FUNCTION_BLOCK "SEQUENCE"   // FB18, GRAPH_PLUS
{ S7_Optimized_Access := 'TRUE' }
VERSION : 0.1
   VAR_INPUT
      OFF_SQ : Bool := false;   // Turn sequence off
      INIT_SQ : Bool := false;   // Set sequence to initial state
      ACK_EF : Bool := false;   // Acknowledge all errors and faults
      S_PREV : Bool := false;   // Output previous step in parameter S_NO
      S_NEXT : Bool := false;   // Indicate next step in parameter S_NO
      SW_AUTO : Bool := false;   // Automatic mode
      SW_TAP : Bool := false;   // Semiautomatic/switch with transition
      SW_TOP : Bool := false;   // Semiautomatic/ignore transition
      SW_MAN : Bool := false;   // Manual mode
      S_SEL : Int := 0;   // Select step to be output to S_NO
      S_ON : Bool := false;   // Activate step indicated in S_NO
      S_OFF : Bool := false;   // Deactivate step indicated S_NO
      T_PUSH : Bool := false;   // Enable transition to switch in semi automatic mode
   END_VAR
   VAR_OUTPUT
      S_NO : Int := 0;   // Step number
      S_MORE : Bool := false;   // More steps are available and can be shown in S_NO
      S_ACTIVE : Bool := false;   // Step indicated in S_NO is active
      ERR_FLT : Bool := false;   // Interlock or supervision group error
      AUTO_ON : Bool := false;   // Automatic mode is active
      TAP_ON : Bool := false;   // Semiautomatic mode/step with transition enabled
      TOP_ON : Bool := false;   // Semiautomatic mode/ignore transition enabled
      MAN_ON : Bool := false;   // Manual mode is active
   END_VAR
   VAR
      HMI_INFO : Array[0..8] of UInt;
      IF_PAR : G7_IfParPlus_V2;
      RT_DATA : G7_RTDataPlus_V2;   // Internal data area
      Trans1 : G7_TransitionPlus_V2;   // Transition structure
      Trans2 : G7_TransitionPlus_V2;   // Transition structure
      Trans3 : G7_TransitionPlus_V2;   // Transition structure
      Trans4 : G7_TransitionPlus_V2;   // Transition structure
      Trans5 : G7_TransitionPlus_V2;   // Transition structure
      Idle : G7_StepPlus_V2;   // Step structure
      Warmup : G7_StepPlus_V2;   // Step structure
      Stabilize : G7_StepPlus_V2;   // Step structure
      Generation : G7_StepPlus_V2;   // Step structure
      CoolDown : G7_StepPlus_V2;   // Step structure
      SINI : Array[0..1] of USInt;
      LSTT : Array[0..4] of USInt;
      ATAJ : Array[0..4] of USInt;
      ATAB : Array[0..4] of USInt;
      PSTT : Array[0..4] of USInt;
      NSTT : Array[0..4] of USInt;
      ASSJ : Array[0..4] of USInt;
      ASSB : Array[0..4] of USInt;
      PTTS : Array[0..4] of USInt;
      NTTS : Array[0..4] of USInt;
      SW_SQTS : Array[0..4] of USInt;
      SWITCH : Array[0..0] of USInt;
      TVX : Array[0..1] of USInt;
      TTX : Array[0..1] of USInt;
      TSX : Array[0..1] of USInt;
      S00X : Array[0..1] of USInt;
      SOFFX : Array[0..1] of USInt;
      SONX : Array[0..1] of USInt;
      SAX : Array[0..1] of USInt;
      SERRX : Array[0..5] of USInt;
      SMX : Array[0..5] of USInt;
      S0X : Array[0..5] of USInt;
      S1X : Array[0..5] of USInt;
      IL_ALARM_INST : Program_Alarm;
      SUP_ALARM_INST : Program_Alarm;
      STEP_TIME_ALARM_INST : Program_Alarm;
      IEC_TIMER_INST : IEC_TIMER;
      TRANSACTION_FLAG : Bool := false;
   END_VAR
   // SINI[0] := 2;
   // SINI[1] := 1;
   // LSTT[0] := 255;
   // LSTT[1] := 255;
   // LSTT[2] := 255;
   // LSTT[4] := 255;
   // ATAJ[1] := 1;
   // ATAJ[2] := 2;
   // ATAJ[3] := 3;
   // ATAJ[4] := 4;
   // ATAB[1] := 1;
   // ATAB[2] := 2;
   // ATAB[3] := 3;
   // ATAB[4] := 4;
   // PSTT[0] := 1;
   // PSTT[1] := 2;
   // PSTT[2] := 3;
   // PSTT[3] := 4;
   // NSTT[0] := 2;
   // NSTT[1] := 3;
   // NSTT[2] := 4;
   // NSTT[4] := 1;
   // ASSJ[1] := 1;
   // ASSJ[2] := 2;
   // ASSJ[3] := 3;
   // ASSJ[4] := 4;
   // ASSB[1] := 1;
   // ASSB[2] := 2;
   // ASSB[3] := 3;
   // ASSB[4] := 4;
   // PTTS[0] := 255;
   // PTTS[1] := 4;
   // PTTS[3] := 1;
   // PTTS[4] := 2;
   // NTTS[0] := 4;
   // NTTS[2] := 1;
   // NTTS[3] := 2;
   // NTTS[4] := 3;
   // TVX[0] := 16#1;
   // TTX[0] := 16#1;
   // TSX[0] := 16#1;
   // S00X[0] := 16#1;
   // SOFFX[0] := 16#1;
   // SONX[0] := 16#1;
   // SAX[0] := 16#1;
   // SERRX[0] := 16#1;
   // SMX[0] := 16#1;
   // S0X[0] := 16#1;
   // S1X[0] := 16#1;
BEGIN
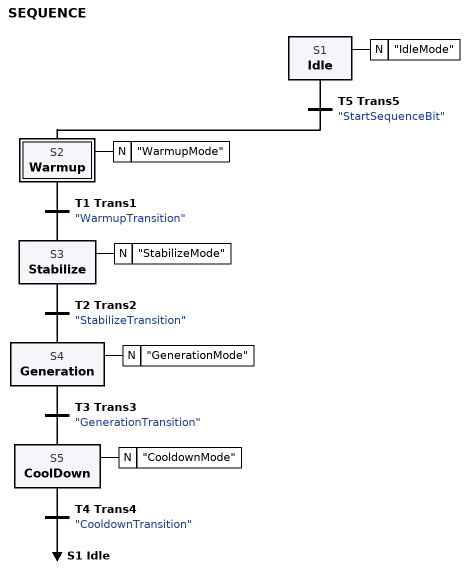
   // sequencer 1
   STEP Idle:   // S1, max time T#10S, warning time T#7S
              N    "IdleMode"
   END_STEP
   TRANSITION Trans5 FROM Idle TO Warmup   // T5
      := "StartSequenceBit";
   END_TRANSITION
   INITIAL_STEP Warmup:   // S2, max time T#10S, warning time T#7S
              N    "WarmupMode"
   END_STEP
   TRANSITION Trans1 FROM Warmup TO Stabilize   // T1
      := "WarmupTransition";
   END_TRANSITION
   STEP Stabilize:   // S3, max time T#10S, warning time T#7S
              N    "StabilizeMode"
   END_STEP
   TRANSITION Trans2 FROM Stabilize TO Generation   // T2
      := "StabilizeTransition";
   END_TRANSITION
   STEP Generation:   // S4, max time T#10S, warning time T#7S
              N    "GenerationMode"
   END_STEP
   TRANSITION Trans3 FROM Generation TO CoolDown   // T3
      := "GenerationTransition";
   END_TRANSITION
   STEP CoolDown:   // S5, max time T#10S, warning time T#7S
              N    "CooldownMode"
   END_STEP
   TRANSITION Trans4 FROM CoolDown TO Idle   // T4, jump
      := "CooldownTransition";
   END_TRANSITION
END_FUNCTION_BLOCK

FUNCTION_BLOCK "HOURMETER_LAD"   // FB19, LAD
{ S7_Optimized_Access := 'TRUE' }
VERSION : 0.1
   VAR
      Accum_elapsed : Time;
      OS1 : Bool;
      MinuteTimedDown : Bool;
      HourCountDown : Bool;
      OS2 : Bool;
      Days_CountedDown : Bool;
      OS3 : Bool;
      OS4 : Bool;
      reset_rto : Bool;
      MinuteCounterreset : Bool;
      Hourcounterreset : Bool;
   END_VAR
   VAR_TEMP
      reset_time : Time;
      reset_HM_Trigger : Bool;
   END_VAR
   VAR_TEMP   // added for the SCL form of the ladder/FBD networks
      _w1 : Bool;
      _w2 : Bool;
      _w3 : Bool;
   END_VAR
BEGIN

REGION Network 1
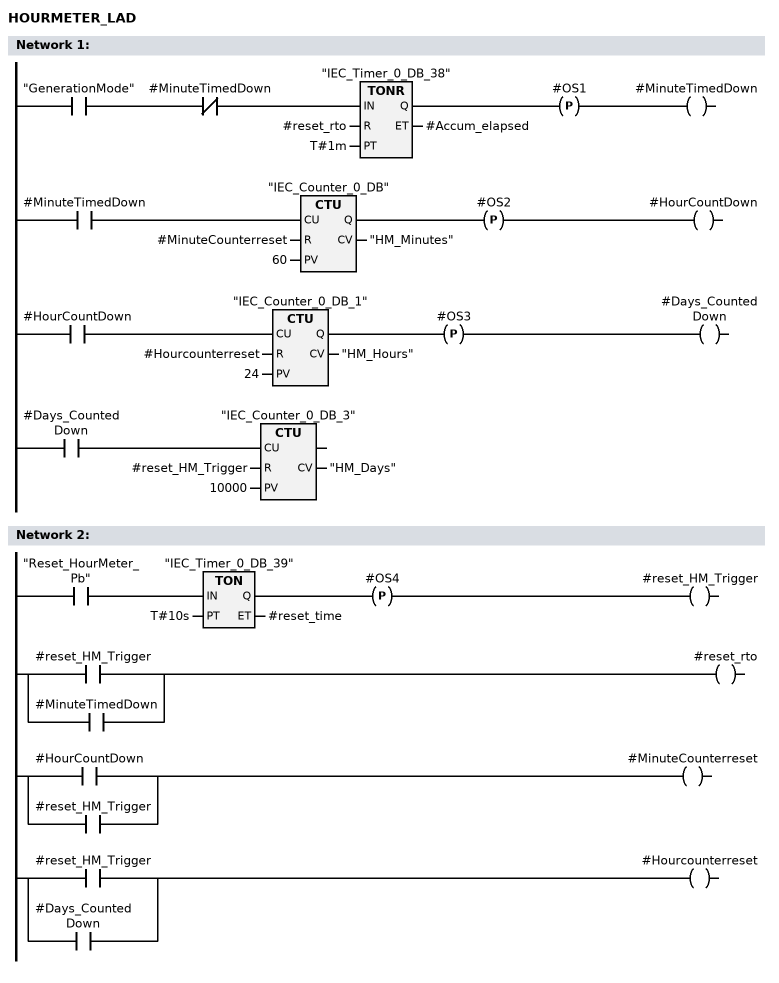
   "IEC_Timer_0_DB_38".TONR(IN := "GenerationMode" AND NOT #MinuteTimedDown,
                           R := #reset_rto,
                           PT := T#1m,
                           ET => #Accum_elapsed);
   #_w1 := "IEC_Timer_0_DB_38".Q AND NOT #OS1;   // rising edge
   #OS1 := "IEC_Timer_0_DB_38".Q;
   #MinuteTimedDown := #_w1;
   "IEC_Counter_0_DB".CTU(CU := #MinuteTimedDown, R := #MinuteCounterreset, PV := 60, CV => "HM_Minutes");
   #_w2 := "IEC_Counter_0_DB".Q AND NOT #OS2;   // rising edge
   #OS2 := "IEC_Counter_0_DB".Q;
   #HourCountDown := #_w2;
   "IEC_Counter_0_DB_1".CTU(CU := #HourCountDown, R := #Hourcounterreset, PV := 24, CV => "HM_Hours");
   #_w3 := "IEC_Counter_0_DB_1".Q AND NOT #OS3;   // rising edge
   #OS3 := "IEC_Counter_0_DB_1".Q;
   #Days_CountedDown := #_w3;
   "IEC_Counter_0_DB_3".CTU(CU := #Days_CountedDown, R := #reset_HM_Trigger, PV := 10000, CV => "HM_Days");
END_REGION

REGION Network 2
   "IEC_Timer_0_DB_39".TON(IN := "Reset_HourMeter_Pb", PT := T#10s, ET => #reset_time);
   #_w1 := "IEC_Timer_0_DB_39".Q AND NOT #OS4;   // rising edge
   #OS4 := "IEC_Timer_0_DB_39".Q;
   #reset_HM_Trigger := #_w1;
   #reset_rto := #reset_HM_Trigger OR #MinuteTimedDown;
   #MinuteCounterreset := #HourCountDown OR #reset_HM_Trigger;
   #Hourcounterreset := #reset_HM_Trigger OR #Days_CountedDown;
END_REGION
END_FUNCTION_BLOCK

FUNCTION_BLOCK "HOURMETER_FBD"   // FB20, FBD
{ S7_Optimized_Access := 'TRUE' }
VERSION : 0.1
   VAR
      Accum_elapsed : Time;
      OS1 : Bool;
      MinuteTimedDown : Bool;
      HourCountDown : Bool;
      OS2 : Bool;
      Days_CountedDown : Bool;
      OS3 : Bool;
      OS4 : Bool;
      reset_rto : Bool;
      MinuteCounterreset : Bool;
      Hourcounterreset : Bool;
   END_VAR
   VAR_TEMP
      reset_time : Time;
      reset_HM_Trigger : Bool;
   END_VAR
   VAR_TEMP   // added for the SCL form of the ladder/FBD networks
      _w1 : Bool;
      _w2 : Bool;
      _w3 : Bool;
   END_VAR
BEGIN

REGION Network 1
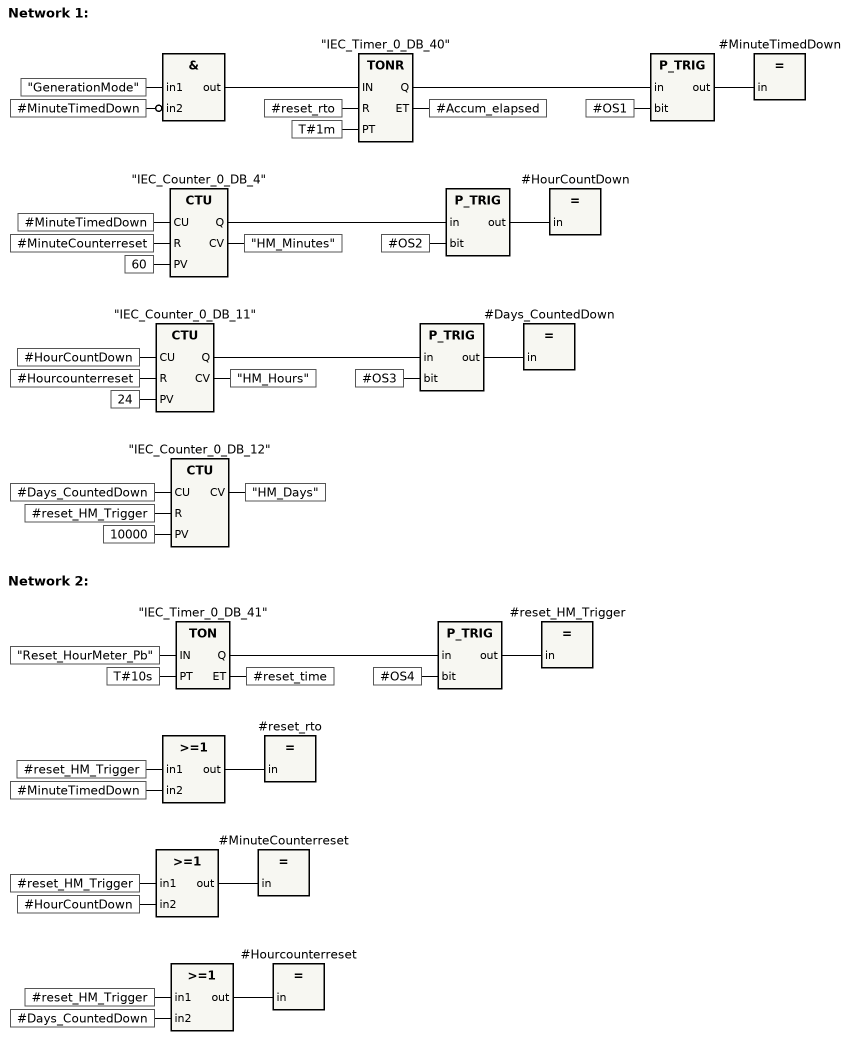
   "IEC_Timer_0_DB_40".TONR(IN := "GenerationMode" AND NOT #MinuteTimedDown,
                           R := #reset_rto,
                           PT := T#1m,
                           ET => #Accum_elapsed);
   #_w1 := "IEC_Timer_0_DB_40".Q AND NOT #OS1;   // rising edge
   #OS1 := "IEC_Timer_0_DB_40".Q;
   #MinuteTimedDown := #_w1;
   "IEC_Counter_0_DB_4".CTU(CU := #MinuteTimedDown, R := #MinuteCounterreset, PV := 60, CV => "HM_Minutes");
   #_w2 := "IEC_Counter_0_DB_4".Q AND NOT #OS2;   // rising edge
   #OS2 := "IEC_Counter_0_DB_4".Q;
   #HourCountDown := #_w2;
   "IEC_Counter_0_DB_11".CTU(CU := #HourCountDown, R := #Hourcounterreset, PV := 24, CV => "HM_Hours");
   #_w3 := "IEC_Counter_0_DB_11".Q AND NOT #OS3;   // rising edge
   #OS3 := "IEC_Counter_0_DB_11".Q;
   #Days_CountedDown := #_w3;
   "IEC_Counter_0_DB_12".CTU(CU := #Days_CountedDown, R := #reset_HM_Trigger, PV := 10000, CV => "HM_Days");
END_REGION

REGION Network 2
   "IEC_Timer_0_DB_41".TON(IN := "Reset_HourMeter_Pb", PT := T#10s, ET => #reset_time);
   #_w1 := "IEC_Timer_0_DB_41".Q AND NOT #OS4;   // rising edge
   #OS4 := "IEC_Timer_0_DB_41".Q;
   #reset_HM_Trigger := #_w1;
   #reset_rto := #reset_HM_Trigger OR #MinuteTimedDown;
   #MinuteCounterreset := #reset_HM_Trigger OR #HourCountDown;
   #Hourcounterreset := #reset_HM_Trigger OR #Days_CountedDown;
END_REGION
END_FUNCTION_BLOCK

FUNCTION_BLOCK "HOURMETER_SCL"   // FB21, SCL
{ S7_Optimized_Access := 'TRUE' }
VERSION : 0.1
   VAR
      Accum_elapsed : Time;
      OS1 : Bool;
      MinuteTimedDown : Bool;
      HourCountDown : Bool;
      OS2 : Bool;
      Days_CountedDown : Bool;
      OS3 : Bool;
      OS4 : Bool;
      reset_rto : Bool;
      MinuteCounterreset : Bool;
      Hourcounterreset : Bool;
   END_VAR
   VAR_TEMP
      reset_time : Time;
      reset_HM_Trigger : Bool;
   END_VAR
BEGIN
   IF "GenerationMode" THEN
    "IEC_Timer_0_DB_42".TONR(IN:=TRUE,
                             R:=#reset_rto,
                             PT:=T#1m,
                             Q=>#MinuteTimedDown,
                             ET=>#Accum_elapsed);
   END_IF;
   IF #MinuteTimedDown THEN
       RESET_TIMER("IEC_Timer_0_DB_42");

   END_IF;


       "IEC_Counter_0_DB_5".CTU(CU:=#MinuteTimedDown,
                               R:=#MinuteCounterreset,
                               PV:=60,
                               Q=>#HourCountDown,
                               CV=>"HM_Minutes");

       "IEC_Counter_0_DB_6".CTU(CU:=#HourCountDown,
                                R:=#Hourcounterreset,
                                PV:=24,
                                Q=>#Days_CountedDown,
                                CV=>"HM_Hours");

   "IEC_Counter_0_DB_7".CTU(CU:=#Days_CountedDown,
                                R:=#reset_HM_Trigger,
                                PV:=10000,
                                CV=>"HM_Days");

   IF "Reset_HourMeter_Pb" THEN
     "IEC_Timer_0_DB_43".TON(IN:=TRUE,
                             PT:=T#10s,
                             Q=>#reset_HM_Trigger,
                             ET=>#reset_time);
   ELSE
       RESET_TIMER("IEC_Timer_0_DB_43");
   END_IF;

   IF #MinuteTimedDown OR #reset_HM_Trigger THEN
       #reset_rto := 1;
   ELSE
       #reset_rto := 0;
   END_IF;


   IF #reset_HM_Trigger OR #HourCountDown THEN
       #MinuteCounterreset := 1;
   ELSE
       #MinuteCounterreset := 0;
   END_IF;

   IF #Days_CountedDown OR #reset_HM_Trigger THEN
       #Hourcounterreset := 1;
   ELSE
       #Hourcounterreset := 0;
   END_IF;
END_FUNCTION_BLOCK

FUNCTION_BLOCK "HOURMETER_STL"   // FB22, STL
{ S7_Optimized_Access := 'TRUE' }
VERSION : 0.1
   VAR
      Accum_elapsed : Time;
      OS1 : Bool;
      MinuteTimedDown : Bool;
      HourCountDown : Bool;
      OS2 : Bool;
      Days_CountedDown : Bool;
      OS3 : Bool;
      OS4 : Bool;
      reset_rto : Bool;
      MinuteCounterreset : Bool;
      Hourcounterreset : Bool;
   END_VAR
   VAR_TEMP
      reset_time : Time;
      reset_HM_Trigger : Bool;
   END_VAR
BEGIN

REGION Network 1
         A     "GenerationMode";
         JC    RTO_timer;
         JU    ResetHM;
   RTO_timer:CALL  TONR , "IEC_Timer_0_DB_44"
         ( IN := TRUE,
           R  := #reset_rto,
           PT := T#1m,
           Q  := #MinuteTimedDown,
           ET := #Accum_elapsed
         );
         CLR;
         A     #MinuteTimedDown;
         JC    Reset_RTO;
         JU    Counters;
   Reset_RTO:CALL  RESET_TIMER
         ( "TIMER" := "IEC_Timer_0_DB_44"
         );

   Counters:CALL  CTU , "IEC_Counter_0_DB_8"
         ( CU := #MinuteTimedDown,
           R  := #MinuteCounterreset,
           PV := 60,
           Q  := #HourCountDown,
           CV := "HM_Minutes"
         );

         CALL  CTU, "IEC_Counter_0_DB_9"
         ( CU := #HourCountDown,
           R  := #Hourcounterreset,
           PV := 24,
           Q  := #Days_CountedDown,
           CV := "HM_Hours"
         );

         CALL  CTU, "IEC_Counter_0_DB_10"
         ( CU := #Days_CountedDown,
           R  := #reset_HM_Trigger,
           PV := 10000,
           Q  := ,
           CV := "HM_Days"
         );

   ResetHM:A     "Reset_HourMeter_Pb";
         JC    set_trigger;
         JU    reset_resetTimer;

   set_trigger:CALL  TON , "IEC_Timer_0_DB_45"
         ( IN := TRUE,
           PT := T#10s,
           Q  := #reset_HM_Trigger,
           ET := #reset_time
         );

         JU    resets;


   reset_resetTimer:CALL  RESET_TIMER
         ( "TIMER" := "IEC_Timer_0_DB_45"
         );
         CLR;
   resets:A     #reset_HM_Trigger;
         O     #MinuteTimedDown;
         =     #reset_rto;
         CLR;
         A     #reset_HM_Trigger;
         O     #HourCountDown;
         =     #MinuteCounterreset;
         CLR;
         A     #reset_HM_Trigger;
         O     #Days_CountedDown;
         =     #Hourcounterreset;
         BE;
END_REGION
END_FUNCTION_BLOCK

FUNCTION "Scale_with_Parameters" : Void   // FC1, FBD
{ S7_Optimized_Access := 'TRUE' }
VERSION : 0.1
   VAR_INPUT
      Input_min : Int;
      Input_signal : Int;
      Input_max : Int;
      Output_max : Int;
      Output_min : Int;
   END_VAR
   VAR_OUTPUT
      sv : Int;
   END_VAR
   VAR_TEMP
      tv : Real;
   END_VAR
BEGIN

REGION Network 1
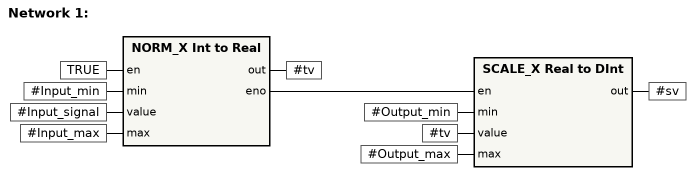
   IF TRUE THEN
       #tv := NORM_X(MIN := #Input_min, VALUE := #Input_signal, MAX := #Input_max);
       #sv := SCALE_X(MIN := #Output_min, VALUE := #tv, MAX := #Output_max);
   END_IF;
END_REGION
END_FUNCTION

FUNCTION "time conversion" : Void   // FC2, FBD
{ S7_Optimized_Access := 'TRUE' }
VERSION : 0.1
   VAR_INPUT
      timein : Int;
   END_VAR
   VAR_OUTPUT
      time_out : Time;
   END_VAR
   VAR_TEMP
      tv1 : Int;
   END_VAR
BEGIN

REGION Network 1
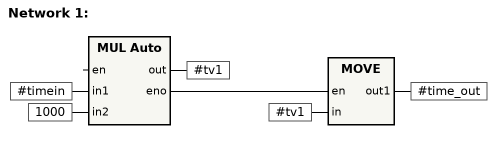
   #tv1 := #timein * 1000;
   #time_out := #tv1;
END_REGION
END_FUNCTION

ORGANIZATION_BLOCK "Main"   // OB1, LAD, ProgramCycle
TITLE = "Main Program Sweep (Cycle)"
{ S7_Optimized_Access := 'TRUE' }
VERSION : 0.1
   VAR_INPUT
      Initial_Call : Bool;   // Initial call of this OB
      Remanence : Bool;   // =True, if remanent data are available
   END_VAR
   VAR_TEMP
      SequenceInit : Bool;
      InitSequence : Bool;
   END_VAR
   VAR_TEMP   // added for the SCL form of the ladder/FBD networks
      _w1 : Bool;
      _w2 : Bool;
      _w3 : Bool;
      _w4 : Bool;
      _w5 : Bool;
      _w6 : Bool;
      _w7 : Bool;
      _w8 : Bool;
      _w9 : Bool;
      _w10 : Bool;
      _w11 : Bool;
      _w12 : Bool;
      _w13 : Bool;
      _w14 : Bool;
   END_VAR
BEGIN

REGION Network 1
   // Simulates the variation of process parameters.
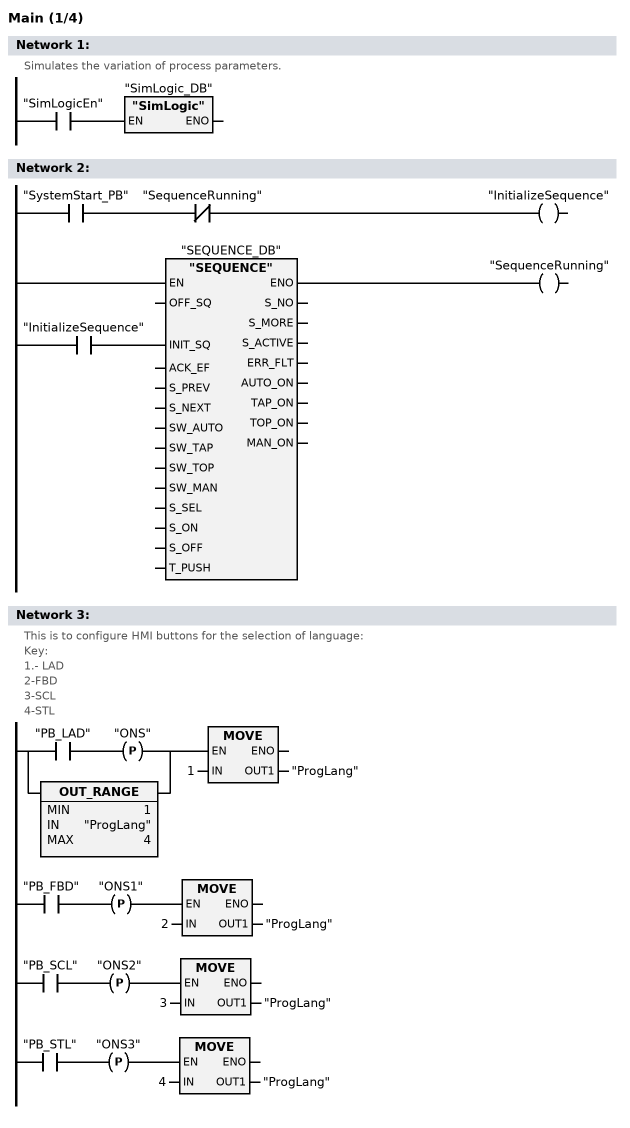
   RUNG wire#powerrail
      Contact( "SimLogicEn" )
      "SimLogic_DB"()
   END_RUNG
   // the same network as SCL:
   IF "SimLogicEn" THEN
       "SimLogic_DB"();   // "SimLogic"
   END_IF;
END_REGION

REGION Network 2
   RUNG wire#powerrail
      Contact( "SystemStart_PB" )
      I_Contact( "SequenceRunning" )
      Coil( "InitializeSequence" )
   END_RUNG
   RUNG wire#powerrail
      "SEQUENCE_DB"(INIT_SQ := wire#w1, OFF_SQ :=, ACK_EF :=, S_PREV :=, S_NEXT :=, SW_AUTO :=, SW_TAP :=, SW_TOP :=, SW_MAN :=, S_SEL :=, S_ON :=, S_OFF :=, T_PUSH :=, S_NO =>, S_MORE =>, S_ACTIVE =>, ERR_FLT =>, AUTO_ON =>, TAP_ON =>, TOP_ON =>, MAN_ON =>)
      Coil( "SequenceRunning" )
   END_RUNG
   RUNG wire#powerrail
      Contact( "InitializeSequence" )
   END_RUNG wire#w1
   // the same network as SCL:
   "InitializeSequence" := "SystemStart_PB" AND NOT "SequenceRunning";
   "SEQUENCE_DB"(INIT_SQ := "InitializeSequence", ENO => #_w1);   // "SEQUENCE"
   "SequenceRunning" := #_w1;
END_REGION

REGION Network 3
   // This is to configure HMI buttons for the selection of language:
   // Key:
   // 1.- LAD
   // 2-FBD
   // 3-SCL
   // 4-STL
   #_w1 := "PB_LAD" AND NOT "ONS";   // rising edge
   "ONS" := "PB_LAD";
   IF #_w1 OR ("ProgLang" < 1) OR ("ProgLang" > 4) THEN "ProgLang" := 1; END_IF;
   #_w2 := "PB_FBD" AND NOT "ONS1";   // rising edge
   "ONS1" := "PB_FBD";
   IF #_w2 THEN "ProgLang" := 2; END_IF;
   #_w3 := "PB_SCL" AND NOT "ONS2";   // rising edge
   "ONS2" := "PB_SCL";
   IF #_w3 THEN "ProgLang" := 3; END_IF;
   #_w4 := "PB_STL" AND NOT "ONS3";   // rising edge
   "ONS3" := "PB_STL";
   IF #_w4 THEN "ProgLang" := 4; END_IF;
END_REGION

REGION Network 4
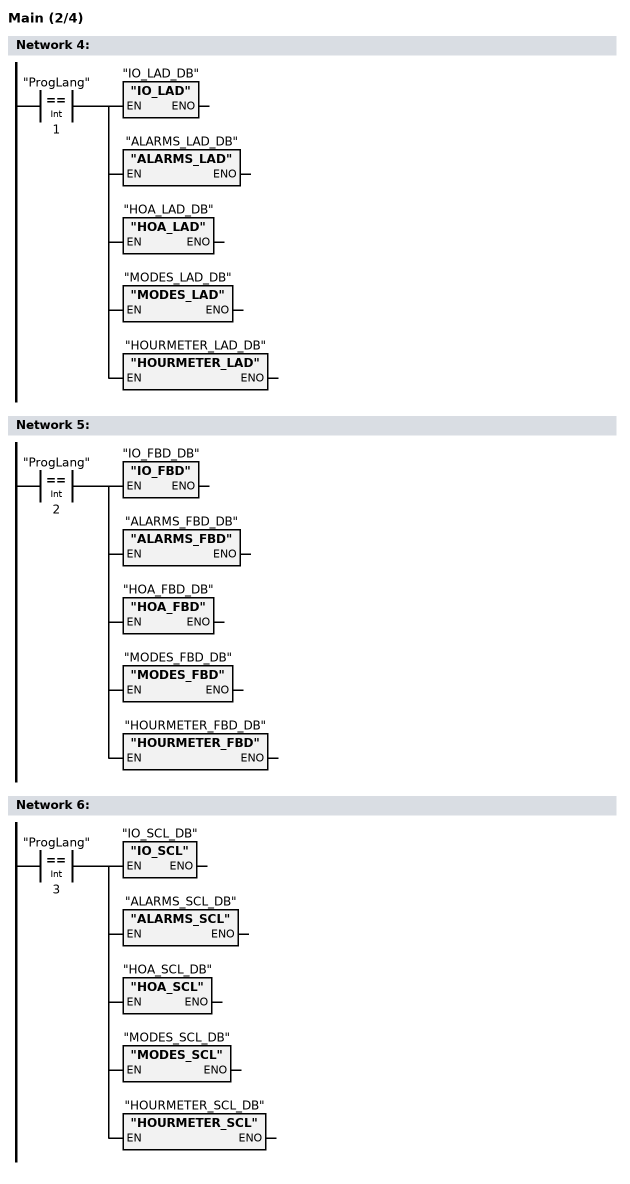
   RUNG wire#powerrail
      { S7_Templates := "SrcType := Int" } EQ_Contact(in1 := "ProgLang", in2 := 1)
      wire#w1
      "IO_LAD_DB"()
   END_RUNG
   RUNG wire#w1
      "ALARMS_LAD_DB"()
   END_RUNG
   RUNG wire#w1
      "HOA_LAD_DB"()
   END_RUNG
   RUNG wire#w1
      "MODES_LAD_DB"()
   END_RUNG
   RUNG wire#w1
      "HOURMETER_LAD_DB"()
   END_RUNG
   // the same network as SCL:
   #_w1 := "ProgLang" = 1;
   IF #_w1 THEN
       "IO_LAD_DB"();   // "IO_LAD"
       "ALARMS_LAD_DB"();   // "ALARMS_LAD"
       "HOA_LAD_DB"();   // "HOA_LAD"
       "MODES_LAD_DB"();   // "MODES_LAD"
       "HOURMETER_LAD_DB"();   // "HOURMETER_LAD"
   END_IF;
END_REGION

REGION Network 5
   RUNG wire#powerrail
      { S7_Templates := "SrcType := Int" } EQ_Contact(in1 := "ProgLang", in2 := 2)
      wire#w1
      "IO_FBD_DB"()
   END_RUNG
   RUNG wire#w1
      "ALARMS_FBD_DB"()
   END_RUNG
   RUNG wire#w1
      "HOA_FBD_DB"()
   END_RUNG
   RUNG wire#w1
      "MODES_FBD_DB"()
   END_RUNG
   RUNG wire#w1
      "HOURMETER_FBD_DB"()
   END_RUNG
   // the same network as SCL:
   #_w1 := "ProgLang" = 2;
   IF #_w1 THEN
       "IO_FBD_DB"();   // "IO_FBD"
       "ALARMS_FBD_DB"();   // "ALARMS_FBD"
       "HOA_FBD_DB"();   // "HOA_FBD"
       "MODES_FBD_DB"();   // "MODES_FBD"
       "HOURMETER_FBD_DB"();   // "HOURMETER_FBD"
   END_IF;
END_REGION

REGION Network 6
   RUNG wire#powerrail
      { S7_Templates := "SrcType := Int" } EQ_Contact(in1 := "ProgLang", in2 := 3)
      wire#w1
      "IO_SCL_DB"()
   END_RUNG
   RUNG wire#w1
      "ALARMS_SCL_DB"()
   END_RUNG
   RUNG wire#w1
      "HOA_SCL_DB"()
   END_RUNG
   RUNG wire#w1
      "MODES_SCL_DB"()
   END_RUNG
   RUNG wire#w1
      "HOURMETER_SCL_DB"()
   END_RUNG
   // the same network as SCL:
   #_w1 := "ProgLang" = 3;
   IF #_w1 THEN
       "IO_SCL_DB"();   // "IO_SCL"
       "ALARMS_SCL_DB"();   // "ALARMS_SCL"
       "HOA_SCL_DB"();   // "HOA_SCL"
       "MODES_SCL_DB"();   // "MODES_SCL"
       "HOURMETER_SCL_DB"();   // "HOURMETER_SCL"
   END_IF;
END_REGION

REGION Network 7
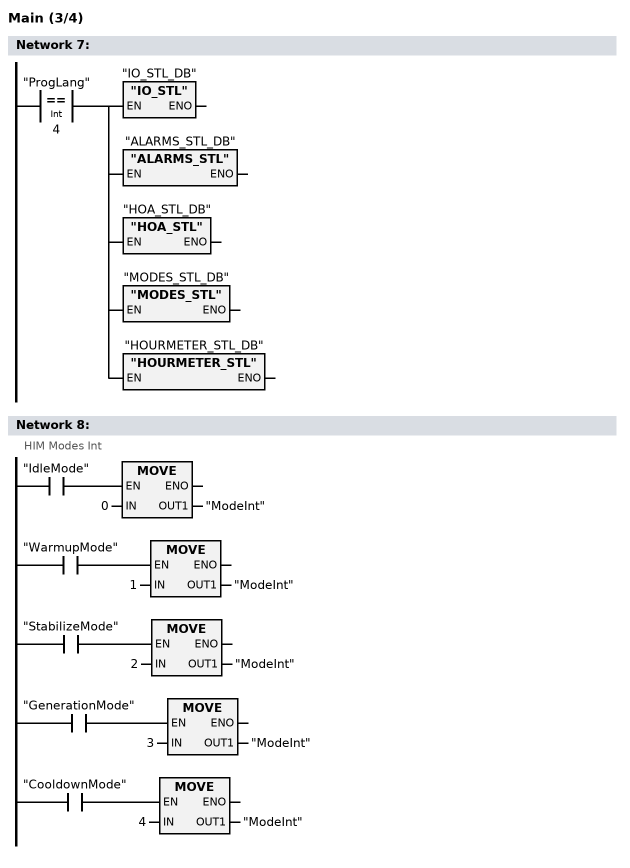
   RUNG wire#powerrail
      { S7_Templates := "SrcType := Int" } EQ_Contact(in1 := "ProgLang", in2 := 4)
      wire#w1
      "IO_STL_DB"()
   END_RUNG
   RUNG wire#w1
      "ALARMS_STL_DB"()
   END_RUNG
   RUNG wire#w1
      "HOA_STL_DB"()
   END_RUNG
   RUNG wire#w1
      "MODES_STL_DB"()
   END_RUNG
   RUNG wire#w1
      "HOURMETER_STL_DB"()
   END_RUNG
   // the same network as SCL:
   #_w1 := "ProgLang" = 4;
   IF #_w1 THEN
       "IO_STL_DB"();   // "IO_STL"
       "ALARMS_STL_DB"();   // "ALARMS_STL"
       "HOA_STL_DB"();   // "HOA_STL"
       "MODES_STL_DB"();   // "MODES_STL"
       "HOURMETER_STL_DB"();   // "HOURMETER_STL"
   END_IF;
END_REGION

REGION Network 8
   // HIM Modes Int
   RUNG wire#powerrail
      Contact( "IdleMode" )
      Move(in := 0, out1 => "ModeInt")
   END_RUNG
   RUNG wire#powerrail
      Contact( "WarmupMode" )
      Move(in := 1, out1 => "ModeInt")
   END_RUNG
   RUNG wire#powerrail
      Contact( "StabilizeMode" )
      Move(in := 2, out1 => "ModeInt")
   END_RUNG
   RUNG wire#powerrail
      Contact( "GenerationMode" )
      Move(in := 3, out1 => "ModeInt")
   END_RUNG
   RUNG wire#powerrail
      Contact( "CooldownMode" )
      Move(in := 4, out1 => "ModeInt")
   END_RUNG
   // the same network as SCL:
   IF "IdleMode" THEN "ModeInt" := 0; END_IF;
   IF "WarmupMode" THEN "ModeInt" := 1; END_IF;
   IF "StabilizeMode" THEN "ModeInt" := 2; END_IF;
   IF "GenerationMode" THEN "ModeInt" := 3; END_IF;
   IF "CooldownMode" THEN "ModeInt" := 4; END_IF;
END_REGION

REGION Network 9
   // Alarm Conversion:
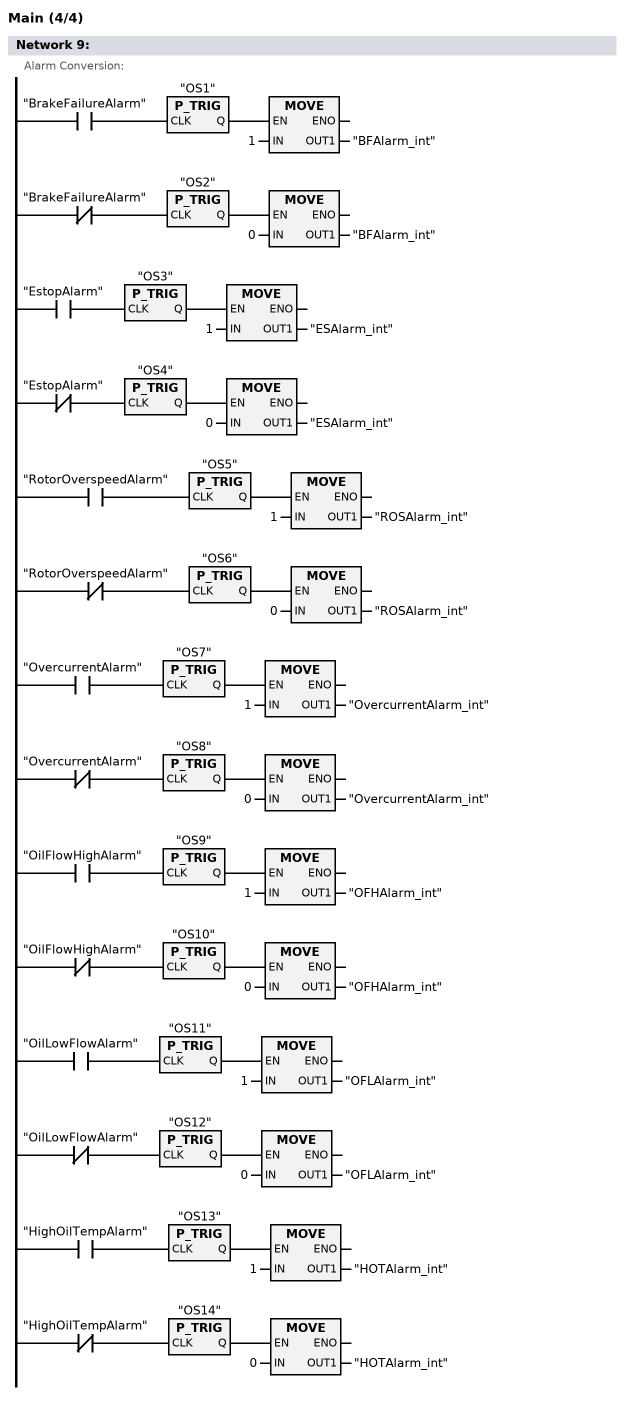
   RUNG wire#powerrail
      Contact( "BrakeFailureAlarm" )
      P_Trig( "OS1" )
      Move(in := 1, out1 => "BFAlarm_int")
   END_RUNG
   RUNG wire#powerrail
      I_Contact( "BrakeFailureAlarm" )
      P_Trig( "OS2" )
      Move(in := 0, out1 => "BFAlarm_int")
   END_RUNG
   RUNG wire#powerrail
      Contact( "EstopAlarm" )
      P_Trig( "OS3" )
      Move(in := 1, out1 => "ESAlarm_int")
   END_RUNG
   RUNG wire#powerrail
      I_Contact( "EstopAlarm" )
      P_Trig( "OS4" )
      Move(in := 0, out1 => "ESAlarm_int")
   END_RUNG
   RUNG wire#powerrail
      Contact( "RotorOverspeedAlarm" )
      P_Trig( "OS5" )
      Move(in := 1, out1 => "ROSAlarm_int")
   END_RUNG
   RUNG wire#powerrail
      I_Contact( "RotorOverspeedAlarm" )
      P_Trig( "OS6" )
      Move(in := 0, out1 => "ROSAlarm_int")
   END_RUNG
   RUNG wire#powerrail
      Contact( "OvercurrentAlarm" )
      P_Trig( "OS7" )
      Move(in := 1, out1 => "OvercurrentAlarm_int")
   END_RUNG
   RUNG wire#powerrail
      I_Contact( "OvercurrentAlarm" )
      P_Trig( "OS8" )
      Move(in := 0, out1 => "OvercurrentAlarm_int")
   END_RUNG
   RUNG wire#powerrail
      Contact( "OilFlowHighAlarm" )
      P_Trig( "OS9" )
      Move(in := 1, out1 => "OFHAlarm_int")
   END_RUNG
   RUNG wire#powerrail
      I_Contact( "OilFlowHighAlarm" )
      P_Trig( "OS10" )
      Move(in := 0, out1 => "OFHAlarm_int")
   END_RUNG
   RUNG wire#powerrail
      Contact( "OilLowFlowAlarm" )
      P_Trig( "OS11" )
      Move(in := 1, out1 => "OFLAlarm_int")
   END_RUNG
   RUNG wire#powerrail
      I_Contact( "OilLowFlowAlarm" )
      P_Trig( "OS12" )
      Move(in := 0, out1 => "OFLAlarm_int")
   END_RUNG
   RUNG wire#powerrail
      Contact( "HighOilTempAlarm" )
      P_Trig( "OS13" )
      Move(in := 1, out1 => "HOTAlarm_int")
   END_RUNG
   RUNG wire#powerrail
      I_Contact( "HighOilTempAlarm" )
      P_Trig( "OS14" )
      Move(in := 0, out1 => "HOTAlarm_int")
   END_RUNG
   // the same network as SCL:
   #_w1 := "BrakeFailureAlarm" AND NOT "OS1";   // rising edge
   "OS1" := "BrakeFailureAlarm";
   IF #_w1 THEN "BFAlarm_int" := 1; END_IF;
   #_w2 := NOT "BrakeFailureAlarm" AND NOT "OS2";   // rising edge
   "OS2" := NOT "BrakeFailureAlarm";
   IF #_w2 THEN "BFAlarm_int" := 0; END_IF;
   #_w3 := "EstopAlarm" AND NOT "OS3";   // rising edge
   "OS3" := "EstopAlarm";
   IF #_w3 THEN "ESAlarm_int" := 1; END_IF;
   #_w4 := NOT "EstopAlarm" AND NOT "OS4";   // rising edge
   "OS4" := NOT "EstopAlarm";
   IF #_w4 THEN "ESAlarm_int" := 0; END_IF;
   #_w5 := "RotorOverspeedAlarm" AND NOT "OS5";   // rising edge
   "OS5" := "RotorOverspeedAlarm";
   IF #_w5 THEN "ROSAlarm_int" := 1; END_IF;
   #_w6 := NOT "RotorOverspeedAlarm" AND NOT "OS6";   // rising edge
   "OS6" := NOT "RotorOverspeedAlarm";
   IF #_w6 THEN "ROSAlarm_int" := 0; END_IF;
   #_w7 := "OvercurrentAlarm" AND NOT "OS7";   // rising edge
   "OS7" := "OvercurrentAlarm";
   IF #_w7 THEN "OvercurrentAlarm_int" := 1; END_IF;
   #_w8 := NOT "OvercurrentAlarm" AND NOT "OS8";   // rising edge
   "OS8" := NOT "OvercurrentAlarm";
   IF #_w8 THEN "OvercurrentAlarm_int" := 0; END_IF;
   #_w9 := "OilFlowHighAlarm" AND NOT "OS9";   // rising edge
   "OS9" := "OilFlowHighAlarm";
   IF #_w9 THEN "OFHAlarm_int" := 1; END_IF;
   #_w10 := NOT "OilFlowHighAlarm" AND NOT "OS10";   // rising edge
   "OS10" := NOT "OilFlowHighAlarm";
   IF #_w10 THEN "OFHAlarm_int" := 0; END_IF;
   #_w11 := "OilLowFlowAlarm" AND NOT "OS11";   // rising edge
   "OS11" := "OilLowFlowAlarm";
   IF #_w11 THEN "OFLAlarm_int" := 1; END_IF;
   #_w12 := NOT "OilLowFlowAlarm" AND NOT "OS12";   // rising edge
   "OS12" := NOT "OilLowFlowAlarm";
   IF #_w12 THEN "OFLAlarm_int" := 0; END_IF;
   #_w13 := "HighOilTempAlarm" AND NOT "OS13";   // rising edge
   "OS13" := "HighOilTempAlarm";
   IF #_w13 THEN "HOTAlarm_int" := 1; END_IF;
   #_w14 := NOT "HighOilTempAlarm" AND NOT "OS14";   // rising edge
   "OS14" := NOT "HighOilTempAlarm";
   IF #_w14 THEN "HOTAlarm_int" := 0; END_IF;
END_REGION
END_ORGANIZATION_BLOCK

ORGANIZATION_BLOCK "PID"   // OB30, LAD, CyclicInterrupt
{ S7_Optimized_Access := 'TRUE' }
VERSION : 0.1
   VAR_INPUT
      Initial_Call : Bool;   // Initial call of this OB
      Event_Count : Int;   // Events discarded
   END_VAR
   VAR_TEMP
      Bsp : Real;
      Vsp : Real;
      BafflehandTrigger : Bool;
      BaffleOffTrigger : Bool;
      VFDhandTrigger : Bool;
      VFDOffTrigger : Bool;
      BaffleAutoTrigger : Bool;
      VFDAutoTrigger : Bool;
   END_VAR
   VAR_TEMP   // added for the SCL form of the ladder/FBD networks
      _w1 : Bool;
      _w2 : Bool;
      _w3 : Bool;
      _w4 : Bool;
      _w5 : Bool;
      _w6 : Bool;
      _w7 : Bool;
   END_VAR
BEGIN

REGION Network 1
   // High Oil flow Alarm Handling:
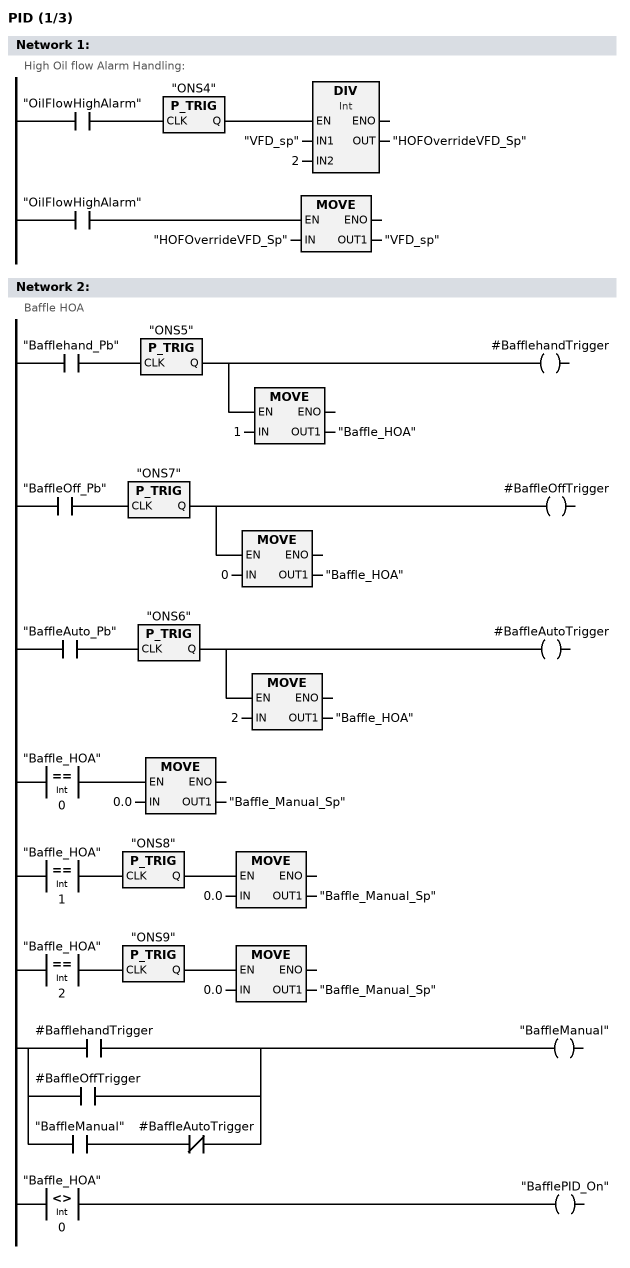
   RUNG wire#powerrail
      Contact( "OilFlowHighAlarm" )
      P_Trig( "ONS4" )
      { S7_Templates := "SrcType := Int" } Div(in1 := "VFD_sp", in2 := 2, out => "HOFOverrideVFD_Sp")
   END_RUNG
   RUNG wire#powerrail
      Contact( "OilFlowHighAlarm" )
      Move(in := "HOFOverrideVFD_Sp", out1 => "VFD_sp")
   END_RUNG
   // the same network as SCL:
   #_w1 := "OilFlowHighAlarm" AND NOT "ONS4";   // rising edge
   "ONS4" := "OilFlowHighAlarm";
   IF #_w1 THEN "HOFOverrideVFD_Sp" := "VFD_sp" / 2; END_IF;
   IF "OilFlowHighAlarm" THEN "VFD_sp" := "HOFOverrideVFD_Sp"; END_IF;
END_REGION

REGION Network 2
   // Baffle HOA
   RUNG wire#powerrail
      Contact( "Bafflehand_Pb" )
      P_Trig( "ONS5" )
      wire#w1
      Coil( #BafflehandTrigger )
   END_RUNG
   RUNG wire#w1
      Move(in := 1, out1 => "Baffle_HOA")
   END_RUNG
   RUNG wire#powerrail
      Contact( "BaffleOff_Pb" )
      P_Trig( "ONS7" )
      wire#w2
      Coil( #BaffleOffTrigger )
   END_RUNG
   RUNG wire#w2
      Move(in := 0, out1 => "Baffle_HOA")
   END_RUNG
   RUNG wire#powerrail
      Contact( "BaffleAuto_Pb" )
      P_Trig( "ONS6" )
      wire#w3
      Coil( #BaffleAutoTrigger )
   END_RUNG
   RUNG wire#w3
      Move(in := 2, out1 => "Baffle_HOA")
   END_RUNG
   RUNG wire#powerrail
      { S7_Templates := "SrcType := Int" } EQ_Contact(in1 := "Baffle_HOA", in2 := 0)
      Move(in := 0.0, out1 => "Baffle_Manual_Sp")
   END_RUNG
   RUNG wire#powerrail
      { S7_Templates := "SrcType := Int" } EQ_Contact(in1 := "Baffle_HOA", in2 := 1)
      P_Trig( "ONS8" )
      Move(in := 0.0, out1 => "Baffle_Manual_Sp")
   END_RUNG
   RUNG wire#powerrail
      { S7_Templates := "SrcType := Int" } EQ_Contact(in1 := "Baffle_HOA", in2 := 2)
      P_Trig( "ONS9" )
      Move(in := 0.0, out1 => "Baffle_Manual_Sp")
   END_RUNG
   RUNG wire#powerrail
      Contact( #BafflehandTrigger )
      wire#w4
      Coil( "BaffleManual" )
   END_RUNG
   RUNG wire#powerrail
      Contact( #BaffleOffTrigger )
   END_RUNG wire#w4
   RUNG wire#powerrail
      Contact( "BaffleManual" )
      I_Contact( #BaffleAutoTrigger )
   END_RUNG wire#w4
   RUNG wire#powerrail
      { S7_Templates := "SrcType := Int" } NE_Contact(in1 := "Baffle_HOA", in2 := 0)
      Coil( "BafflePID_On" )
   END_RUNG
   // the same network as SCL:
   #_w1 := "Bafflehand_Pb" AND NOT "ONS5";   // rising edge
   "ONS5" := "Bafflehand_Pb";
   #BafflehandTrigger := #_w1;
   IF #_w1 THEN "Baffle_HOA" := 1; END_IF;
   #_w2 := "BaffleOff_Pb" AND NOT "ONS7";   // rising edge
   "ONS7" := "BaffleOff_Pb";
   #BaffleOffTrigger := #_w2;
   IF #_w2 THEN "Baffle_HOA" := 0; END_IF;
   #_w3 := "BaffleAuto_Pb" AND NOT "ONS6";   // rising edge
   "ONS6" := "BaffleAuto_Pb";
   #BaffleAutoTrigger := #_w3;
   IF #_w3 THEN "Baffle_HOA" := 2; END_IF;
   IF "Baffle_HOA" = 0 THEN "Baffle_Manual_Sp" := 0.0; END_IF;
   #_w4 := "Baffle_HOA" = 1;
   #_w5 := #_w4 AND NOT "ONS8";   // rising edge
   "ONS8" := #_w4;
   IF #_w5 THEN "Baffle_Manual_Sp" := 0.0; END_IF;
   #_w6 := "Baffle_HOA" = 2;
   #_w7 := #_w6 AND NOT "ONS9";   // rising edge
   "ONS9" := #_w6;
   IF #_w7 THEN "Baffle_Manual_Sp" := 0.0; END_IF;
   "BaffleManual" := #BafflehandTrigger OR #BaffleOffTrigger OR ("BaffleManual" AND NOT #BaffleAutoTrigger);
   "BafflePID_On" := "Baffle_HOA" <> 0;
END_REGION

REGION Network 3
   // VFD HOA
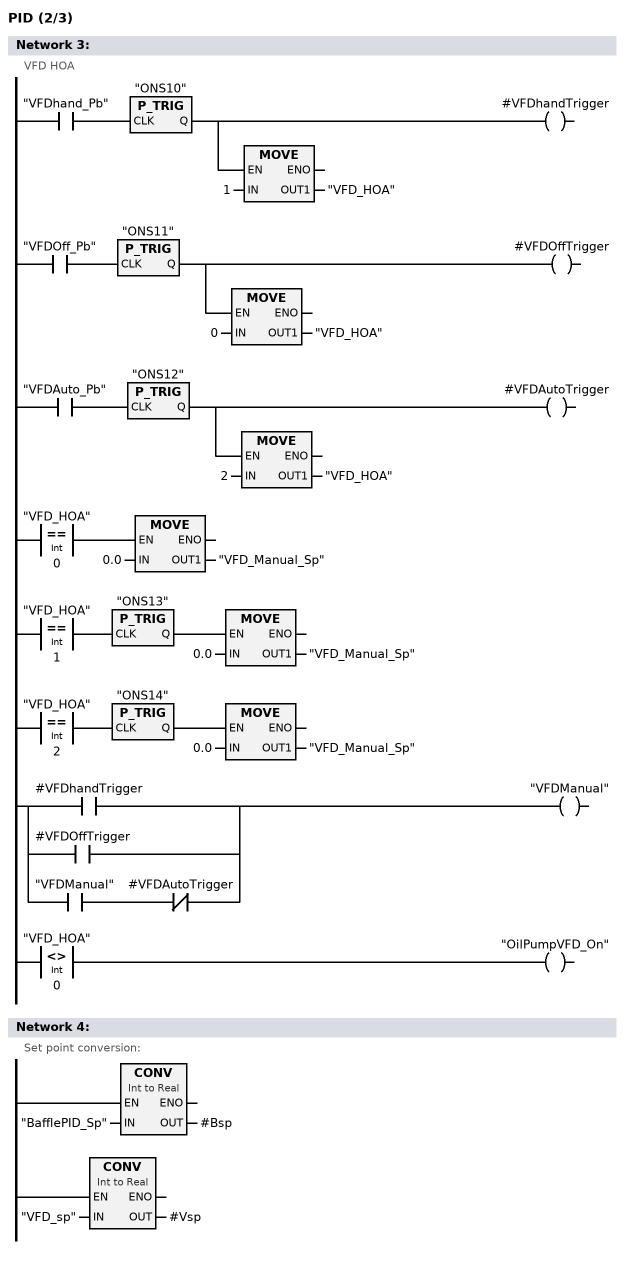
   RUNG wire#powerrail
      Contact( "VFDhand_Pb" )
      P_Trig( "ONS10" )
      wire#w1
      Coil( #VFDhandTrigger )
   END_RUNG
   RUNG wire#w1
      Move(in := 1, out1 => "VFD_HOA")
   END_RUNG
   RUNG wire#powerrail
      Contact( "VFDOff_Pb" )
      P_Trig( "ONS11" )
      wire#w2
      Coil( #VFDOffTrigger )
   END_RUNG
   RUNG wire#w2
      Move(in := 0, out1 => "VFD_HOA")
   END_RUNG
   RUNG wire#powerrail
      Contact( "VFDAuto_Pb" )
      P_Trig( "ONS12" )
      wire#w3
      Coil( #VFDAutoTrigger )
   END_RUNG
   RUNG wire#w3
      Move(in := 2, out1 => "VFD_HOA")
   END_RUNG
   RUNG wire#powerrail
      { S7_Templates := "SrcType := Int" } EQ_Contact(in1 := "VFD_HOA", in2 := 0)
      Move(in := 0.0, out1 => "VFD_Manual_Sp")
   END_RUNG
   RUNG wire#powerrail
      { S7_Templates := "SrcType := Int" } EQ_Contact(in1 := "VFD_HOA", in2 := 1)
      P_Trig( "ONS13" )
      Move(in := 0.0, out1 => "VFD_Manual_Sp")
   END_RUNG
   RUNG wire#powerrail
      { S7_Templates := "SrcType := Int" } EQ_Contact(in1 := "VFD_HOA", in2 := 2)
      P_Trig( "ONS14" )
      Move(in := 0.0, out1 => "VFD_Manual_Sp")
   END_RUNG
   RUNG wire#powerrail
      Contact( #VFDhandTrigger )
      wire#w4
      Coil( "VFDManual" )
   END_RUNG
   RUNG wire#powerrail
      Contact( #VFDOffTrigger )
   END_RUNG wire#w4
   RUNG wire#powerrail
      Contact( "VFDManual" )
      I_Contact( #VFDAutoTrigger )
   END_RUNG wire#w4
   RUNG wire#powerrail
      { S7_Templates := "SrcType := Int" } NE_Contact(in1 := "VFD_HOA", in2 := 0)
      Coil( "OilPumpVFD_On" )
   END_RUNG
   // the same network as SCL:
   #_w1 := "VFDhand_Pb" AND NOT "ONS10";   // rising edge
   "ONS10" := "VFDhand_Pb";
   #VFDhandTrigger := #_w1;
   IF #_w1 THEN "VFD_HOA" := 1; END_IF;
   #_w2 := "VFDOff_Pb" AND NOT "ONS11";   // rising edge
   "ONS11" := "VFDOff_Pb";
   #VFDOffTrigger := #_w2;
   IF #_w2 THEN "VFD_HOA" := 0; END_IF;
   #_w3 := "VFDAuto_Pb" AND NOT "ONS12";   // rising edge
   "ONS12" := "VFDAuto_Pb";
   #VFDAutoTrigger := #_w3;
   IF #_w3 THEN "VFD_HOA" := 2; END_IF;
   IF "VFD_HOA" = 0 THEN "VFD_Manual_Sp" := 0.0; END_IF;
   #_w4 := "VFD_HOA" = 1;
   #_w5 := #_w4 AND NOT "ONS13";   // rising edge
   "ONS13" := #_w4;
   IF #_w5 THEN "VFD_Manual_Sp" := 0.0; END_IF;
   #_w6 := "VFD_HOA" = 2;
   #_w7 := #_w6 AND NOT "ONS14";   // rising edge
   "ONS14" := #_w6;
   IF #_w7 THEN "VFD_Manual_Sp" := 0.0; END_IF;
   "VFDManual" := #VFDhandTrigger OR #VFDOffTrigger OR ("VFDManual" AND NOT #VFDAutoTrigger);
   "OilPumpVFD_On" := "VFD_HOA" <> 0;
END_REGION

REGION Network 4
   // Set point conversion:
   RUNG wire#powerrail
      { S7_Templates := "[SrcType := Int, DestType := Real]" } Convert(in := "BafflePID_Sp", out => #Bsp)
   END_RUNG
   RUNG wire#powerrail
      { S7_Templates := "[SrcType := Int, DestType := Real]" } Convert(in := "VFD_sp", out => #Vsp)
   END_RUNG
   // the same network as SCL:
   #Bsp := INT_TO_REAL("BafflePID_Sp");
   #Vsp := INT_TO_REAL("VFD_sp");
END_REGION

REGION Network 5
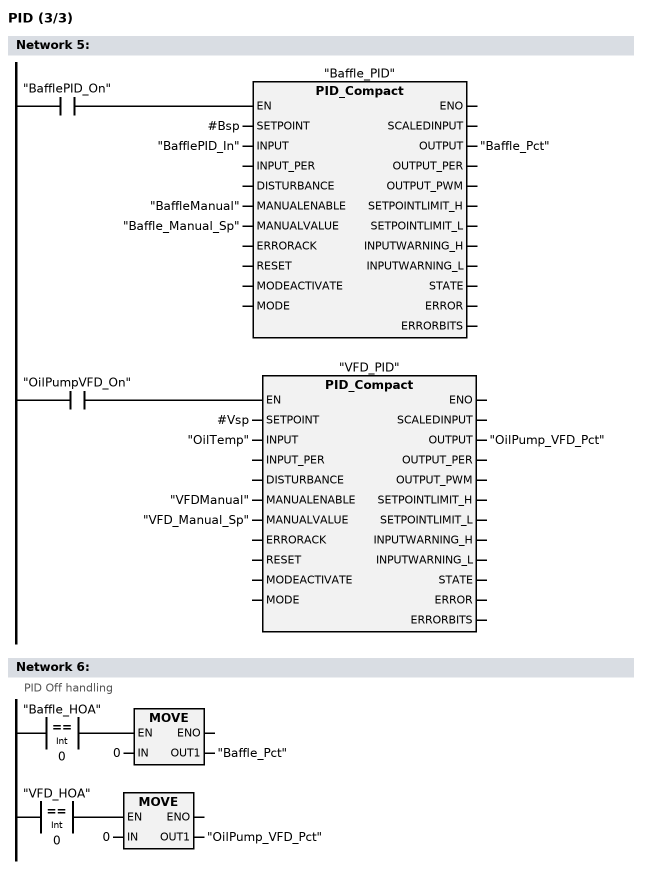
   IF "BafflePID_On" THEN
       "Baffle_PID"(Setpoint := #Bsp,   // PID_Compact
                    Input := "BafflePID_In",
                    ManualEnable := "BaffleManual",
                    ManualValue := "Baffle_Manual_Sp",
                    Output => "Baffle_Pct");
   END_IF;
   IF "OilPumpVFD_On" THEN
       "VFD_PID"(Setpoint := #Vsp,   // PID_Compact
                 Input := "OilTemp",
                 ManualEnable := "VFDManual",
                 ManualValue := "VFD_Manual_Sp",
                 Output => "OilPump_VFD_Pct");
   END_IF;
END_REGION

REGION Network 6
   // PID Off handling
   RUNG wire#powerrail
      { S7_Templates := "SrcType := Int" } EQ_Contact(in1 := "Baffle_HOA", in2 := 0)
      Move(in := 0, out1 => "Baffle_Pct")
   END_RUNG
   RUNG wire#powerrail
      { S7_Templates := "SrcType := Int" } EQ_Contact(in1 := "VFD_HOA", in2 := 0)
      Move(in := 0, out1 => "OilPump_VFD_Pct")
   END_RUNG
   // the same network as SCL:
   IF "Baffle_HOA" = 0 THEN "Baffle_Pct" := 0; END_IF;
   IF "VFD_HOA" = 0 THEN "OilPump_VFD_Pct" := 0; END_IF;
END_REGION
END_ORGANIZATION_BLOCK

(* ===== HMI "HMI_RT_1" =====
system functions are stored by id; their names below are inferred from use
connection "1500 PLC": ETHERNET, S7_1500_OMS

HMI tags "Default tag table"
   "SystemStartPb" : Bool = PLC SystemStart_PB AT %M39.1, 1 s
   "SystemStopPb" : Bool = PLC SystemStop_PB AT %M39.4, 1 s
   "EstopAlarm" : Int = PLC ESAlarm_int AT %MW118, 1 s
   "BrakefailureAlarm" : Int = PLC BFAlarm_int AT %MW116, 1 s
   "LowOilFlowAlarm" : Int = PLC OFLAlarm_int AT %MW126, 1 s
   "HighOilFlowAlarm" : Int = PLC OFHAlarm_int AT %MW124, 1 s
   "HighOiltempAlarm" : Int = PLC HOTAlarm_int AT %MW128, 1 s
   "OverspeedAlarm" : Int = PLC ROSAlarm_int AT %MW120, 1 s
   "OvercurrentAlarm" : Int = PLC OvercurrentAlarm_int AT %MW122, 1 s
   "AlarmReset" : Bool = PLC AlarmReset AT %M31.6, 1 s
   "AlarmSilence" : Bool = PLC AlarmSilence AT %M31.7, 1 s
   "BrakeEn" : Bool = PLC Brake_Out AT %M0.0, 1 s
   "StationIntEn" : Bool = PLC StationInterlock_Out AT %M1.4, 1 s
   "VFDEn" : Bool = PLC OilPumpVFDen_Out AT %M0.2, 1 s
   "BaffleEn" : Int = PLC Baffle_Out AT %MW18, 1 s
   "AlarmHornEn" : Bool = PLC AlarmHorn_Out AT %M1.3, 1 s
   "BrakeHandPb" : Bool = PLC Brake_hand_Pb AT %M30.2, 1 s
   "BrakeOffPb" : Bool = PLC Brake_Off_Pb AT %M30.1, 1 s
   "BrakeAutoPb" : Bool = PLC Brake_Auto_Pb AT %M30.3, 1 s
   "StatInthandPb" : Bool = PLC StationInterlock_Hand_Pb AT %M31.0, 1 s
   "StatIntOffPb" : Bool = PLC StationInterlock_Off_Pb AT %M30.7, 1 s
   "StatIntAutoPb" : Bool = PLC StationInterlock_Auto_Pb AT %M31.1, 1 s
   "VFDhandPb" : Bool = PLC VFDhand_Pb AT %M95.2, 1 s
   "VFDOffPb" : Bool = PLC VFDOff_Pb AT %M95.3, 1 s
   "VFDAutoPb" : Bool = PLC VFDAuto_Pb AT %M95.4, 1 s
   "Bafflehandpb" : Bool = PLC Bafflehand_Pb AT %M94.0, 1 s
   "BaffleOffPb" : Bool = PLC BaffleOff_Pb AT %M94.3, 1 s
   "BaffleAutoPb" : Bool = PLC BaffleAuto_Pb AT %M94.1, 1 s
   "AlarmHornHandPb" : Bool = PLC AlarmHorn_Hand_Pb AT %M30.5, 1 s
   "AlarmHornOffPb" : Bool = PLC AlarmHorn_Off_Pb AT %M30.4, 1 s
   "AlarmHornAutoPb" : Bool = PLC AlarmHorn_Auto_Pb AT %M30.6, 1 s
   "ModeInt" : Int = PLC ModeInt AT %MW114, 1 s
   "AlarmHornHOA" : Int = PLC AlarmHorn_HOA AT %MW34, 1 s
   "BaffleHOA" : Int = PLC Baffle_HOA AT %MW40, 1 s
   "StationInterlockHOA" : Int = PLC StationInterlock_HOA AT %MW36, 1 s
   "VFDHOA" : Int = PLC VFD_HOA AT %MW106, 1 s
   "BrakeHOA" : Int = PLC Brake_HOA AT %MW32, 1 s
   "BrakefailureDelay" : Int = PLC BrakeFailureDelaySpt AT %MW64, 1 s
   "Overcurrentdelay" : Int = PLC OvercurrentDelaySpt AT %MW46, 1 s
   "OvercurrentSp" : Int = PLC Overcurrent_Sp AT %MW48, 1 s
   "OverspeedDelay" : Int = PLC RotorOverpeedDelaySpt AT %MW54, 1 s
   "OverspeedSp" : Int = PLC RotorSpeed_Sp AT %MW56, 1 s
   "HighOilTempSp" : Int = PLC HighOilTemp_Sp AT %MW52, 1 s
   "HighOilTempDelay" : Int = PLC HighOilTempDelaySpt AT %MW50, 1 s
   "HighOilFlowdelay" : Int = PLC OilFlowHighDelaySpt AT %MW58, 1 s
   "HighOilFlowSp" : Int = PLC OilFlowhigh_Sp AT %MW62, 1 s
   "LowOilFlowDelay" : Int = PLC OilLowFlowDelaySpt AT %MW60, 1 s
   "LowOilFlowSp" : Int = PLC OilLowFlow_Sp AT %MW44, 1 s
   "WarmupOilTemp" : Int = PLC WarmupOilTemp AT %MW74, 1 s
   "WarmupDelay" : Int = PLC WarmupOilDelay_Sp AT %MW76, 1 s
   "StabilizeDelay" : Int = PLC StabilizeDelay_Sp AT %MW86, 1 s
   "CurrentSp" : Int = PLC StabilizeKW_Sp AT %MW82, 1 s
   "WarmupVFDPct" : Int = PLC Warmup_VFD_Pct AT %MW110, 1 s
   "CoolDownOilTemp" : Int = PLC CooldownOiltemp_Sp AT %MW90, 1 s
   "CoolDownDelay" : Int = PLC CooldownDelay_Sp AT %MW88, 1 s
   "HM_Minutes" : Int = PLC HM_Minutes AT %MW28, 1 s
   "HM_Hours" : Int = PLC HM_Hours AT %MW108, 1 s
   "HM_Days" : Int = PLC HM_Days AT %MW112, 1 s
   "HM_ResetPb" : Bool = PLC Reset_HourMeter_Pb AT %M72.1, 1 s
   "Faultmode" : Bool = PLC FaultMode AT %M38.4, 1 s
   "VFDManualSp" : Real = PLC VFD_Manual_Sp AT %MD102, 1 s
   "BaffleManualSp" : Real = PLC Baffle_Manual_Sp AT %MD96, 1 s
   "ProgLang" : Int = PLC ProgLang AT %MW12, 1 s
   "PB_LAD" : Bool = PLC PB_LAD AT %M0.3, 1 s
   "PB_FBD" : Bool = PLC PB_FBD AT %M0.5, 1 s
   "PB_SCL" : Bool = PLC PB_SCL AT %M0.6, 1 s
   "PB_STL" : Bool = PLC PB_STL AT %M0.7, 1 s
   "Current" : Int = PLC Current AT %MW26, 1 s
   "OilTemp" : Int = PLC OilTemp AT %MW20, 1 s
   "OilFlow" : Int = PLC OilFlow AT %MW22, 1 s
   "VFDPct" : Int = PLC OilPump_VFD_Pct AT %MW14, 1 s
   "BafflePct" : Int = PLC Baffle_Pct AT %MW16, 1 s
   "RPM" : Int = PLC RPM AT %MW24, 1 s
   "EstopPB" : Bool = PLC Estop AT %M43.4, 1 s

discrete alarms
   1: 'Estop open', class Errors, trigger "EstopAlarm" bit 0
   2: 'Brake Failed', class Errors, trigger "BrakefailureAlarm" bit 0
   3: 'Overcurrent', class Errors, trigger "OvercurrentAlarm" bit 0
   4: 'Rotor overspeed', class Errors, trigger "OverspeedAlarm" bit 0
   5: 'Oil Low Flow', class Errors, trigger "LowOilFlowAlarm" bit 0
   6: 'High Oil Flow', class Errors, trigger "HighOilFlowAlarm" bit 0
   7: 'High Oil Temp', class Errors, trigger "HighOiltempAlarm" bit 0

screen "Alarms" 600x800
   Button "Button_5" at 20,327 size 96x32; TextOff 'Main'
      on Click: ActivateScreen("Status", 0)
   Button "Button_6" at 139,327 size 96x32; TextOff 'Overview'
      on Click: ActivateScreen("Overview", 0)
   Button "Button_7" at 258,327 size 96x32; TextOff 'Alarms'
      on Click: ActivateScreen("Alarms", 0)
   Button "Button_8" at 377,327 size 96x32; TextOff 'Config'
      on Click: ActivateScreen("Config", 0)
   Circle "Circle_4" at 514,322 size 60x60
      Visibility <- "Faultmode"
   TextField "Text field_1" at 12,13 size 210x29; Text 'Alarm Management'
   AlarmView "Alarm view_1" at 0,42 size 599x198
   Button "Button_9" at 334,250 size 119x42; TextOff 'RESET'
      on Release: ResetBit("AlarmReset")
      on Press: SetBit("AlarmReset")
   Button "Button_1" at 473,249 size 119x42; TextOff 'SLIENCE'
      on Release: ResetBit("AlarmSilence")
      on Press: SetBit("AlarmSilence")
   Group "Group" at 8,250 size 36x36
   Group "Group_1" at 53,250 size 38x36
   Group "Group_2" at 98,250 size 38x36
   Group "Group_3" at 143,250 size 37x36
   Group "Group_4" at 188,250 size 39x36
   Group "Group_5" at 228,250 size 41x36
   Group "Group_6" at 278,249 size 44x36
   Button "Button_11" at 552,0 size 48x43; TextOff 'ESTOP'
      on Release: ResetBit("EstopPB")
      on Press: SetBit("EstopPB")
   TextField "Text field_9" at 528,340 size 27x22; Text 'OK'
      Visibility <- "Faultmode"
   TextField "Text field_10" at 514,340 size 54x22; Text 'Alarm!'
      Visibility <- "Faultmode"
   Circle "Circle_1" at 8,250 size 36x36
      Visibility <- "EstopAlarm"
   TextField "Text field_2" at 11,262 size 33x15; Text 'EStop'
      Visibility <- "EstopAlarm"
   Circle "Circle_2" at 53,250 size 36x36
      Visibility <- "BrakefailureAlarm"
   TextField "Text field_3" at 56,262 size 35x15; Text 'Brake'
      Visibility <- "BrakefailureAlarm"
   Circle "Circle_5" at 98,250 size 36x36
      Visibility <- "OverspeedAlarm"
   TextField "Text field_4" at 101,262 size 35x15; Text 'Speed'
      Visibility <- "OverspeedAlarm"
   Circle "Circle_6" at 143,250 size 36x36
      Visibility <- "LowOilFlowAlarm"
   TextField "Text field_5" at 146,262 size 34x15; Text 'LFlow'
      Visibility <- "LowOilFlowAlarm"
   Circle "Circle_7" at 188,250 size 36x36
      Visibility <- "HighOilFlowAlarm"
   TextField "Text field_6" at 191,262 size 36x15; Text 'HFlow'
      Visibility <- "HighOilFlowAlarm"
   Circle "Circle_8" at 233,250 size 36x36
      Visibility <- "HighOiltempAlarm"
   TextField "Text field_7" at 228,262 size 41x15; Text 'HTemp'
      Visibility <- "HighOiltempAlarm"
   Circle "Circle_9" at 283,249 size 36x36
      Visibility <- "OvercurrentAlarm"
   TextField "Text field_8" at 278,261 size 44x15; Text 'Current'
      Visibility <- "OvercurrentAlarm"

screen "Config" 600x800
   TextField "Text field_1" at 8,8 size 148x29; Text 'Configuration'
   IOField "I/O field_1" at 150,59 size 96x32; FormatPattern s99999
      ProcessValue <- "WarmupOilTemp"
   TextField "Text field_2" at 8,63 size 117x23; Text 'Warmup Temp:'
   TextField "Text field_3" at 8,37 size 129x24; Text 'process values:'
   IOField "I/O field_2" at 151,95 size 96x32; FormatPattern s99999
      ProcessValue <- "WarmupDelay"
   TextField "Text field_4" at 9,99 size 115x23; Text 'Warmup Delay:'
   IOField "I/O field_3" at 152,131 size 96x32; FormatPattern s99999
      ProcessValue <- "CurrentSp"
   TextField "Text field_5" at 10,135 size 97x23; Text 'Current(Kw):'
   IOField "I/O field_4" at 153,167 size 96x32; FormatPattern s99999
      ProcessValue <- "StabilizeDelay"
   TextField "Text field_6" at 11,171 size 113x23; Text 'Stabilize Delay:'
   IOField "I/O field_5" at 154,203 size 96x32; FormatPattern s99999
      ProcessValue <- "CoolDownOilTemp"
   TextField "Text field_7" at 12,207 size 130x23; Text 'CoolDown Temp:'
   IOField "I/O field_6" at 155,239 size 96x32; FormatPattern s99999
      ProcessValue <- "CoolDownDelay"
   TextField "Text field_8" at 13,243 size 128x23; Text 'CoolDown Delay:'
   IOField "I/O field_7" at 449,52 size 96x32; FormatPattern s99999
      ProcessValue <- "BrakefailureDelay"
   TextField "Text field_9" at 280,56 size 135x23; Text 'Brake failure delay'
   IOField "I/O field_8" at 450,88 size 96x32; FormatPattern s99999
      ProcessValue <- "OverspeedSp"
   TextField "Text field_10" at 308,92 size 122x23; Text 'Overspeed RPM:'
   IOField "I/O field_9" at 451,124 size 96x32; FormatPattern s99999
      ProcessValue <- "OverspeedDelay"
   TextField "Text field_11" at 292,128 size 130x23; Text 'Overspeed Delay:'
   IOField "I/O field_10" at 452,160 size 96x32; FormatPattern s99999
      ProcessValue <- "HighOilTempSp"
   TextField "Text field_12" at 280,164 size 148x23; Text 'OverTemp Degrees:'
   IOField "I/O field_11" at 453,196 size 96x32; FormatPattern s99999
      ProcessValue <- "LowOilFlowSp"
   TextField "Text field_13" at 311,200 size 115x23; Text 'Low Flow GPM:'
   IOField "I/O field_12" at 454,232 size 96x32; FormatPattern s99999
      ProcessValue <- "LowOilFlowDelay"
   TextField "Text field_14" at 312,236 size 122x23; Text 'Low Flow Delay:'
   TextField "Text field_15" at 274,36 size 124x24; Text 'Alarm Values :'
   IOField "I/O field_13" at 452,272 size 96x32; FormatPattern s99999
      ProcessValue <- "HighOilFlowSp"
   TextField "Text field_16" at 310,276 size 119x23; Text 'High Flow GPM:'
   IOField "I/O field_14" at 453,308 size 96x32; FormatPattern s99999
      ProcessValue <- "HighOilFlowdelay"
   TextField "Text field_17" at 311,312 size 126x23; Text 'High Flow Delay:'
   IOField "I/O field_15" at 451,348 size 96x32; FormatPattern s99999
      ProcessValue <- "HighOilTempDelay"
   TextField "Text field_18" at 304,352 size 130x23; Text 'OverTemp Delay:'
   Button "Button_5" at 14,687 size 96x32; TextOff 'Main'
      on Click: ActivateScreen("Status", 0)
   Button "Button_6" at 133,687 size 96x32; TextOff 'Overview'
      on Click: ActivateScreen("Overview", 0)
   Button "Button_7" at 252,687 size 96x32; TextOff 'Alarms'
      on Click: ActivateScreen("Alarms", 0)
   Button "Button_8" at 371,687 size 96x32; TextOff 'Config'
      on Click: ActivateScreen("Config", 0)
   TextField "Text field_19" at 73,317 size 117x24; Text 'HOA controls:'
   TextField "Text field_20" at 75,335 size 94x24; Text 'Alarm Horn:'
   Button "Button_1" at 72,365 size 34x25; TextOff 'H'
      on Press: SetBit("AlarmHornHandPb")
      on Release: ResetBit("AlarmHornHandPb")
   Button "Button_2" at 112,365 size 34x25; TextOff 'O'
      on Release: ResetBit("AlarmHornOffPb")
      on Press: SetBit("AlarmHornOffPb")
   Button "Button_3" at 152,365 size 34x25; TextOff 'A'
      on Release: ResetBit("AlarmHornAutoPb")
      on Press: SetBit("AlarmHornAutoPb")
   TextField "Text field_21" at 73,397 size 50x23; Text 'Brake:'
   Button "Button_4" at 76,420 size 34x25; TextOff 'H'
      on Release: ResetBit("BrakeHandPb")
      on Press: SetBit("BrakeHandPb")
   Button "Button_9" at 116,420 size 34x25; TextOff 'O'
      on Release: ResetBit("BrakeOffPb")
      on Press: SetBit("BrakeOffPb")
   Button "Button_10" at 156,420 size 34x25; TextOff 'A'
      on Release: ResetBit("BrakeAutoPb")
      on Press: SetBit("BrakeAutoPb")
   TextField "Text field_22" at 72,446 size 125x23; Text 'Station interlock:'
   Button "Button_11" at 78,471 size 34x25; TextOff 'H'
      on Release: ResetBit("StatInthandPb")
      on Press: SetBit("StatInthandPb")
   Button "Button_12" at 118,471 size 34x25; TextOff 'O'
      on Release: ResetBit("StatIntOffPb")
      on Press: SetBit("StatIntOffPb")
   Button "Button_13" at 158,471 size 34x25; TextOff 'A'
      on Release: ResetBit("StatIntAutoPb")
      on Press: SetBit("StatIntAutoPb")
   Button "Button_14" at 70,525 size 34x25; TextOff 'H'
      on Release: ResetBit("Bafflehandpb")
      on Press: SetBit("Bafflehandpb")
   Button "Button_15" at 107,525 size 34x25; TextOff 'O'
      on Release: ResetBit("BaffleOffPb")
      on Press: SetBit("BaffleOffPb")
   Button "Button_16" at 150,525 size 34x25; TextOff 'A'
      on Release: ResetBit("BaffleAutoPb")
      on Press: SetBit("BaffleAutoPb")
   Button "Button_17" at 77,585 size 34x25; TextOff 'H'
      on Release: ResetBit("VFDhandPb")
      on Press: SetBit("VFDhandPb")
   Button "Button_18" at 118,586 size 34x25; TextOff 'O'
      on Release: ResetBit("VFDOffPb")
      on Press: SetBit("VFDOffPb")
   Button "Button_19" at 158,586 size 34x25; TextOff 'A'
      on Release: ResetBit("VFDAutoPb")
      on Press: SetBit("VFDAutoPb")
   TextField "Text field_23" at 72,499 size 50x23; Text 'Baffle:'
   TextField "Text field_24" at 70,555 size 106x23; Text 'OilPump VFD:'
   Rectangle "Rectangle_3" at 195,363 size 28x27
      Visibility <- "AlarmHornHOA"
   Rectangle "Rectangle_4" at 195,363 size 28x27
      Visibility <- "AlarmHornHOA"
   Rectangle "Rectangle_5" at 195,363 size 28x27
      Visibility <- "AlarmHornHOA"
   Rectangle "Rectangle_6" at 195,522 size 28x27
      Visibility <- "BaffleHOA"
   Rectangle "Rectangle_7" at 195,522 size 28x27
      Visibility <- "BaffleHOA"
   Rectangle "Rectangle_8" at 195,522 size 28x27
      Visibility <- "BaffleHOA"
   Rectangle "Rectangle_9" at 199,585 size 28x27
      Visibility <- "VFDHOA"
   Rectangle "Rectangle_10" at 199,585 size 28x27
      Visibility <- "VFDHOA"
   Rectangle "Rectangle_11" at 199,584 size 28x27
      Visibility <- "VFDHOA"
   Rectangle "Rectangle_12" at 196,469 size 28x27
      Visibility <- "StationInterlockHOA"
   Rectangle "Rectangle_13" at 196,470 size 28x27
      Visibility <- "StationInterlockHOA"
   Rectangle "Rectangle_14" at 196,469 size 28x27
      Visibility <- "StationInterlockHOA"
   Rectangle "Rectangle_15" at 192,421 size 28x27
      Visibility <- "BrakeHOA"
   Rectangle "Rectangle_16" at 193,421 size 28x27
      Visibility <- "BrakeHOA"
   Rectangle "Rectangle_17" at 194,420 size 28x27
      Visibility <- "BrakeHOA"
   IOField "I/O field_16" at 479,523 size 96x32; FormatPattern s999999999.999
      ProcessValue <- "BaffleManualSp"
   IOField "I/O field_17" at 477,595 size 96x32; FormatPattern s999999999.999
      ProcessValue <- "VFDManualSp"
   TextField "Text field_25" at 286,525 size 168x23; Text 'Baffle Manual Setpoint:'
   TextField "Text field_26" at 264,593 size 190x23; Text 'OilPump Manual Setpoint:'
   TextField "Text field_27" at 278,390 size 142x23; Text 'OverCurrent Delay:'
   IOField "I/O field_18" at 454,388 size 96x32; FormatPattern s99999
      ProcessValue <- "Overcurrentdelay"
   IOField "I/O field_19" at 457,428 size 96x32; FormatPattern s99999
      ProcessValue <- "OvercurrentSp"
   TextField "Text field_28" at 271,428 size 166x23; Text 'OverCurrent Set point:'
   IOField "I/O field_20" at 156,275 size 96x32; FormatPattern s99999
      ProcessValue <- "WarmupVFDPct"
   TextField "Text field_30" at 16,276 size 121x23; Text 'WarmupVFD %:'
   Button "Button_20" at 545,0 size 55x37; TextOff 'ESTOP'
      on Release: ResetBit("EstopPB")
      on Press: SetBit("EstopPB")
   Circle "Circle_4" at 530,669 size 60x60
      Visibility <- "Faultmode"
   TextField "Text field_29" at 544,687 size 27x22; Text 'OK'
      Visibility <- "Faultmode"
   TextField "Text field_31" at 530,687 size 54x22; Text 'Alarm!'
      Visibility <- "Faultmode"

screen "Overview" 600x800
   Button "Button_5" at 18,376 size 96x32; TextOff 'Main'
      on Click: ActivateScreen("Status", 0)
   Button "Button_6" at 137,376 size 96x32; TextOff 'Overview'
      on Click: ActivateScreen("Overview", 0)
   Button "Button_7" at 256,376 size 96x32; TextOff 'Alarms'
      on Click: ActivateScreen("Alarms", 0)
   Button "Button_8" at 375,376 size 96x32; TextOff 'Config'
      on Click: ActivateScreen("Config", 0)
   TextField "Text field_1" at 8,8 size 186x29; Text 'System Overview'
   TextField "Text field_2" at 395,131 size 15x22; Text 'Text'
   GraphicView "Graphic view_1" at 13,8 size 563x271; Picture "Annotation 2020-07-19 180952"
   IOField "I/O field_1" at 7,257 size 96x32; FormatPattern s99999
      ProcessValue <- "BafflePct"
   TextField "Text field_3" at 16,288 size 62x22; Text 'Baffle %'
   IOField "I/O field_2" at 269,253 size 96x32; FormatPattern s99999
      ProcessValue <- "RPM"
   TextField "Text field_4" at 295,289 size 34x22; Text 'RPM'
   IOField "I/O field_3" at 339,76 size 96x32; FormatPattern s99999
      ProcessValue <- "VFDPct"
   TextField "Text field_5" at 365,55 size 52x22; Text 'VFD %'
   TextField "Text field_6" at 25,121 size 47x22; Text 'Baffle'
   TextField "Text field_7" at 126,131 size 78x22; Text 'AlarmHorn'
   TextField "Text field_8" at 8,8 size 15x22; Text 'Text'
   TextField "Text field_9" at 391,114 size 35x22; Text 'VFD'
   TextField "Text field_10" at 453,33 size 98x22; Text 'power Station'
   TextField "Text field_11" at 16,16 size 83x23; Text 'Overview:'
   Group "Group" at 244,209 size 147x35
   Group "Group_1" at 244,208 size 147x35
   Group "Group_2" at 398,158 size 193x35
   Group "Group_3" at 398,158 size 193x35
   Group "Group_4" at 9,48 size 36x36
   Group "Group_5" at 54,48 size 38x36
   Group "Group_6" at 99,48 size 38x36
   Group "Group_7" at 144,48 size 37x36
   Group "Group_8" at 189,48 size 39x36
   Group "Group_9" at 229,48 size 41x36
   Group "Group_10" at 279,47 size 44x36
   TextField "Text field_23" at 151,327 size 109x29; Text 'Idle Mode'
      Visibility <- "ModeInt"
   TextField "Text field_24" at 151,327 size 158x29; Text 'Warmup Mode'
      Visibility <- "ModeInt"
   TextField "Text field_25" at 151,327 size 157x29; Text 'Stabilize Mode'
      Visibility <- "ModeInt"
   TextField "Text field_26" at 152,327 size 184x29; Text 'Generation Mode'
      Visibility <- "ModeInt"
   TextField "Text field_27" at 151,327 size 175x29; Text 'CoolDown Mode'
      Visibility <- "ModeInt"
   IOField "I/O field_4" at 339,26 size 96x32; FormatPattern s99999
      ProcessValue <- "OilTemp"
   TextField "Text field_28" at 346,4 size 64x22; Text 'Oil Temp'
   IOField "I/O field_5" at 469,302 size 96x32; FormatPattern s99999
      ProcessValue <- "Current"
   TextField "Text field_30" at 392,310 size 58x22; Text 'Current:'
   Button "Button_11" at 550,0 size 50x38; TextOff 'ESTOP'
      on Release: ResetBit("EstopPB")
      on Press: SetBit("EstopPB")
   Circle "Circle_4" at 516,351 size 60x60
      Visibility <- "Faultmode"
   TextField "Text field_29" at 530,369 size 27x22; Text 'OK'
      Visibility <- "Faultmode"
   TextField "Text field_31" at 516,369 size 54x22; Text 'Alarm!'
      Visibility <- "Faultmode"
   Rectangle "Rectangle_1" at 244,209 size 147x35
      Visibility <- "BrakeEn"
   TextField "Text field_12" at 261,212 size 116x22; Text 'Brake Engaged'
      Visibility <- "BrakeEn"
   Rectangle "Rectangle_2" at 244,208 size 147x35
      Visibility <- "BrakeEn"
   TextField "Text field_13" at 253,212 size 122x22; Text 'Brake Released'
      Visibility <- "BrakeEn"
   Rectangle "Rectangle_4" at 398,158 size 193x35
      Visibility <- "StationIntEn"
   TextField "Text field_15" at 413,163 size 165x22; Text 'Interlock Disengaged'
      Visibility <- "StationIntEn"
   Rectangle "Rectangle_5" at 398,158 size 193x35
      Visibility <- "StationIntEn"
   TextField "Text field_14" at 414,165 size 141x22; Text 'Interlock Engaged'
      Visibility <- "StationIntEn"
   Circle "Circle_1" at 9,48 size 36x36
      Visibility <- "EstopAlarm"
   TextField "Text field_16" at 12,60 size 33x15; Text 'EStop'
      Visibility <- "EstopAlarm"
   Circle "Circle_2" at 54,48 size 36x36
      Visibility <- "BrakefailureAlarm"
   TextField "Text field_17" at 57,60 size 35x15; Text 'Brake'
      Visibility <- "BrakefailureAlarm"
   Circle "Circle_5" at 99,48 size 36x36
      Visibility <- "OverspeedAlarm"
   TextField "Text field_18" at 102,60 size 35x15; Text 'Speed'
      Visibility <- "OverspeedAlarm"
   Circle "Circle_6" at 144,48 size 36x36
      Visibility <- "LowOilFlowAlarm"
   TextField "Text field_19" at 147,60 size 34x15; Text 'LFlow'
      Visibility <- "LowOilFlowAlarm"
   Circle "Circle_7" at 189,48 size 36x36
      Visibility <- "HighOilFlowAlarm"
   TextField "Text field_20" at 192,60 size 36x15; Text 'HFlow'
      Visibility <- "HighOilFlowAlarm"
   Circle "Circle_8" at 234,48 size 36x36
      Visibility <- "HighOiltempAlarm"
   TextField "Text field_21" at 229,60 size 41x15; Text 'HTemp'
      Visibility <- "HighOiltempAlarm"
   Circle "Circle_9" at 284,47 size 36x36
      Visibility <- "OvercurrentAlarm"
   TextField "Text field_22" at 279,59 size 44x15; Text 'Current'
      Visibility <- "OvercurrentAlarm"

screen "Status" 600x800
   TextField "Text field_17" at 328,215 size 96x29; Text 'OFFLINE'
   Button "Button_5" at 20,327 size 96x32; TextOff 'Main'
      on Click: ActivateScreen("Status", 0)
   Button "Button_6" at 139,327 size 96x32; TextOff 'Overview'
      on Click: ActivateScreen("Overview", 0)
   Button "Button_7" at 258,327 size 96x32; TextOff 'Alarms'
      on Click: ActivateScreen("Alarms", 0)
   Button "Button_8" at 377,327 size 96x32; TextOff 'Config'
      on Click: ActivateScreen("Config", 0)
   TextField "Text field_1" at 8,8 size 164x29; Text 'System Status'
   TextField "Text field_2" at 410,79 size 109x29; Text 'Idle Mode'
      Visibility <- "ModeInt"
   TextField "Text field_3" at 410,79 size 158x29; Text 'Warmup Mode'
      Visibility <- "ModeInt"
   TextField "Text field_4" at 410,79 size 157x29; Text 'Stabilize Mode'
      Visibility <- "ModeInt"
   TextField "Text field_5" at 411,79 size 184x29; Text 'Generation Mode'
      Visibility <- "ModeInt"
   TextField "Text field_6" at 410,79 size 175x29; Text 'CoolDown Mode'
      Visibility <- "ModeInt"
   TextField "Text field_7" at 424,124 size 83x29; Text 'Ladder'
      Visibility <- "ProgLang"
   Button "Button_1" at 22,278 size 96x32; TextOff 'LAD'
      on Press: SetBit("PB_LAD")
      on Release: ResetBit("PB_LAD")
   Button "Button_2" at 165,282 size 96x32; TextOff 'FBD'
      on Release: ResetBit("PB_FBD")
      on Press: SetBit("PB_FBD")
   Button "Button_3" at 328,282 size 96x32; TextOff 'SCL'
      on Release: ResetBit("PB_SCL")
      on Press: SetBit("PB_SCL")
   Button "Button_4" at 491,282 size 96x32; TextOff 'STL'
      on Release: ResetBit("PB_STL")
      on Press: SetBit("PB_STL")
   TextField "Text field_8" at 389,124 size 199x29; Text 'Structured Control'
      Visibility <- "ProgLang"
   TextField "Text field_9" at 424,124 size 170x29; Text 'Statement Lists'
      Visibility <- "ProgLang"
   TextField "Text field_10" at 411,123 size 169x29; Text 'Function Blocks'
      Visibility <- "ProgLang"
   Button "Button_9" at 3,37 size 227x56; TextOff 'START'
      on Press: SetBit("SystemStartPb")
      on Release: ResetBit("SystemStartPb")
   Button "Button_10" at 3,93 size 225x64; TextOff 'STOP'
      on Press: SetBit("SystemStopPb")
      on Release: ResetBit("SystemStopPb")
   IOField "I/O field_1" at 297,167 size 96x32; FormatPattern s99999
      ProcessValue <- "Current"
   TextField "Text field_11" at 208,170 size 83x29; Text 'Current:'
   TextField "Text field_12" at 392,170 size 42x29; Text 'KW'
   TextField "Text field_13" at 213,215 size 94x29; Text 'Interlock:'
   TextField "Text field_14" at 326,215 size 109x29; Text 'ENGAGED'
      Visibility <- "StationIntEn"
   TextField "Text field_15" at 24,186 size 19x29; Text 'Text'
   Button "Button_11" at 540,0 size 60x48; TextOff 'ESTOP'
      on Release: ResetBit("EstopPB")
      on Press: SetBit("EstopPB")
   Circle "Circle_4" at 514,322 size 60x60
      Visibility <- "Faultmode"
   TextField "Text field_16" at 528,340 size 27x22; Text 'OK'
      Visibility <- "Faultmode"
   TextField "Text field_18" at 514,340 size 54x22; Text 'Alarm!'
      Visibility <- "Faultmode"
*)